FUNCTION_BLOCK FB_DiscreteValve EXTENDS FB_Actor2Point
VAR_INPUT
END_VAR
VAR_OUTPUT
END_VAR
VAR
	//I/O Links
	bValveIsOpen: BOOL; //True if valve is (actual) open
END_VAR

//Outputs
//Output (On/Off) := bSetStatusOn;

SelectControlMode();
SetState();

PROPERTY bWorking : BOOL; //TRUE if valve is (actual) open
GET
bWorking := bValveIsOpen;
END_GET
END_PROPERTY

METHOD SetState //Set opc ua states
VAR_INPUT
END_VAR
controlState.bStatusOn := bWorking;
END_METHOD

END_FUNCTION_BLOCK

(* stored: Version 1.1.0.1, ProductVersion 3.1.4024.9
   POU FB_DiscreteValve: Id {7c2d056e-b7a5-47e0-8780-c9ad927c4f52}, SpecialFunc None
   Property bWorking: Id {cdbb5f1b-344d-4814-8f11-6e79cecb4130}
   Get Get: Id {5a2e688a-3a5b-4624-bb4a-7ac0319686e3}
   Method SetState: Id {eeff4fab-f10d-4347-b3e3-7e5a71f7ad61} *)
